// TIA Portal V17 export
// export: Created 2024-06-14T09:53:18.6441466Z, ExportSetting WithDefaults, DisplayName Totally Integrated Automation Portal, DisplayVersion V17, DisplayName TIA Portal Openness, DisplayVersion V17, DisplayName TIA Portal Version Control Interface, DisplayVersion V17, DisplayName Simotion SCOUT TIA, DisplayVersion 5.4.3.0, DisplayName SINAMICS Startdrive Advanced, DisplayVersion V17 SP1 Update 1, DisplayName SINAMICS Startdrive G110M, G120, G120C, G120D, G120P, G115D, DisplayVersion V17 SP1 Update 1, DisplayName SINAMICS Startdrive G130, G150, S120, S150, SINAMICS MV, S210, DisplayVersion V17 SP1 Update 1, DisplayName STEP 7 Professional, DisplayVersion V17, DisplayName STEP 7 Safety, DisplayVersion V17, DisplayName WinCC Professional, DisplayVersion V17
DATA_BLOCK "MB_CLIENT_DB_L1S4"   // DB7
// stored: AutoNumber true, DBAccessibleFromOPCUA true, InstanceOfName MB_CLIENT, OfSystemLibElement MB_CLIENT, OfSystemLibVersion 5.1
"MB_CLIENT"
   // VAR_INPUT
   //    REQ : Bool;
   //    DISCONNECT : Bool;
   //    MB_MODE : USInt;
   //    MB_DATA_ADDR : UDInt;
   //    MB_DATA_LEN : UInt;
   // END_VAR
   // VAR_OUTPUT
   //    DONE : Bool;
   //    BUSY : Bool;
   //    ERROR : Bool;
   //    STATUS { ExternalVisible := 'False'} : Word;
   // END_VAR
   // VAR_IN_OUT
   //    MB_DATA_PTR : Variant;
   //    CONNECT : Variant;
   // END_VAR
   // VAR
   //    TCON { S7_SetPoint := 'True'} : TCON;
   //    TDISCON { S7_SetPoint := 'True'} : TDISCON;
   //    TSEND { S7_SetPoint := 'True'} : TSEND;
   //    TRECEIVE { S7_SetPoint := 'True'} : TRCV;
   //    TRESET { S7_SetPoint := 'True'} : T_RESET;
   //    TDIAG { S7_SetPoint := 'True'} : T_DIAG;
   //    TDIAG_Status { S7_SetPoint := 'True'} : TDiag_Status;
   //    Blocked_Proc_Timeout : Real;
   //    Rcv_Timeout : Real;
   //    MB_Unit_ID : Byte;
   //    MB_Transaction_ID : Word;
   //    MB_State { ExternalWritable := 'False'} : Word;
   //    SAVED_MB_DATA_ADDR : UDInt;
   //    SAVED_DATA_LEN : UInt;
   //    SAVED_MB_MODE : USInt;
   //    Connection_ID : Word;
   //    Retries : Word;
   //    TEMP_DATA { ExternalWritable := 'False'} : Array[1..263] of Byte;
   //    rcv_timer { ExternalAccessible := 'False'; ExternalVisible := 'False'; ExternalWritable := 'False'; S7_SetPoint := 'True'} : TON_TIME;
   //    wd_timer { ExternalAccessible := 'False'; ExternalVisible := 'False'; ExternalWritable := 'False'; S7_SetPoint := 'True'} : TON_TIME;
   //    Connected : Bool;
   //    Active { ExternalWritable := 'False'} : Bool;
   // END_VAR
BEGIN
END_DATA_BLOCK
